FUNCTION_BLOCK P_Join (* Parallel gateway join: EO once the first N branch inputs have all arrived *)
  (* Standard: 61499-2 *)
  (* Version 2.0, 2026-09-27, Project contributors, Filling cell reference model *)
  PACKAGE fillingcell;
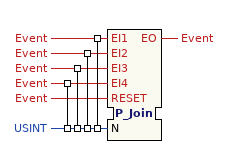
  EVENT_INPUT
    EI1 WITH N;
    EI2 WITH N;
    EI3 WITH N;
    EI4 WITH N;
    RESET;
  END_EVENT
  EVENT_OUTPUT
    EO;
  END_EVENT
  VAR_INPUT
    N : USINT := 2;
  END_VAR
  VAR
    A1 : BOOL;
    A2 : BOOL;
    A3 : BOOL;
    A4 : BOOL;
    Arrived : USINT;
  END_VAR
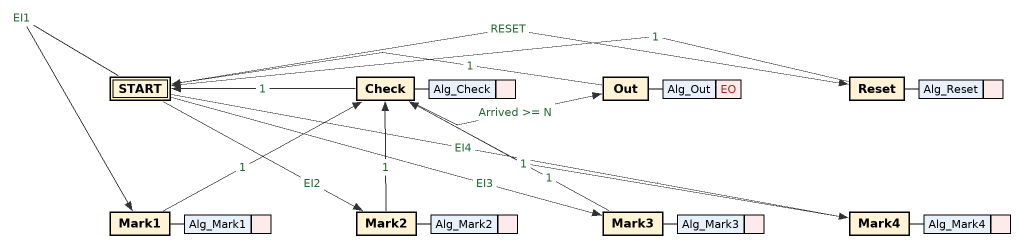
  EC_STATES
    START;
    Check : Alg_Check;
    Out : Alg_Out -> EO;
    Reset : Alg_Reset;
    Mark1 : Alg_Mark1;
    Mark2 : Alg_Mark2;
    Mark3 : Alg_Mark3;
    Mark4 : Alg_Mark4;
  END_STATES
  EC_TRANSITIONS
    START TO Mark1 := EI1;
    Mark1 TO Check := 1;
    START TO Mark2 := EI2;
    Mark2 TO Check := 1;
    START TO Mark3 := EI3;
    Mark3 TO Check := 1;
    START TO Mark4 := EI4;
    Mark4 TO Check := 1;
    Check TO Out := Arrived >= N;
    Check TO START := 1;
    Out TO START := 1;
    START TO Reset := RESET;
    Reset TO START := 1;
  END_TRANSITIONS
  ALGORITHM Alg_Check IN ST:
Arrived := 0;
IF A1 THEN Arrived := Arrived + 1; END_IF;
IF A2 THEN Arrived := Arrived + 1; END_IF;
IF A3 THEN Arrived := Arrived + 1; END_IF;
IF A4 THEN Arrived := Arrived + 1; END_IF;
  END_ALGORITHM
  ALGORITHM Alg_Out IN ST:
A1 := FALSE;
A2 := FALSE;
A3 := FALSE;
A4 := FALSE;
  END_ALGORITHM
  ALGORITHM Alg_Reset IN ST:
A1 := FALSE;
A2 := FALSE;
A3 := FALSE;
A4 := FALSE;
  END_ALGORITHM
  ALGORITHM Alg_Mark1 IN ST:
A1 := TRUE;
  END_ALGORITHM
  ALGORITHM Alg_Mark2 IN ST:
A2 := TRUE;
  END_ALGORITHM
  ALGORITHM Alg_Mark3 IN ST:
A3 := TRUE;
  END_ALGORITHM
  ALGORITHM Alg_Mark4 IN ST:
A4 := TRUE;
  END_ALGORITHM
END_FUNCTION_BLOCK
